FUNCTION_BLOCK p12_controlLight
VAR_INPUT
	button: BOOL;
END_VAR
VAR_OUTPUT
	light: BOOL;
END_VAR
VAR
	positiveEdgeDetection: R_TRIG;
	buttonPulse: BOOL;
	memoryCell: SR;
END_VAR

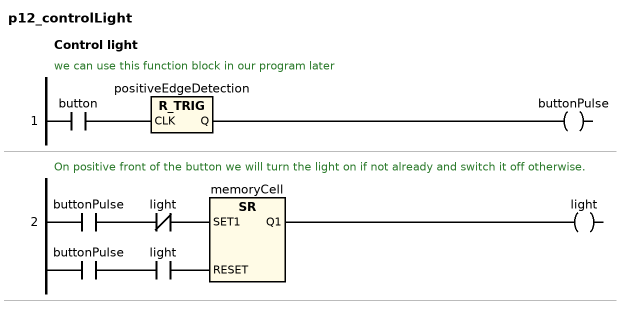
// NETWORK 1: Control light
// we can use this function block in our program later
positiveEdgeDetection(CLK := button); // R_TRIG
buttonPulse := positiveEdgeDetection.Q;

// NETWORK 2
// On positive front of the button we will turn the light on if not already and switch it off otherwise.
memoryCell(SET1 := buttonPulse AND NOT light, RESET := buttonPulse AND light); // SR
light := memoryCell.Q1;

END_FUNCTION_BLOCK

(* stored: Version 1.1.0.1, ProductVersion 3.1.4024.13
   POU p12_controlLight: Id {7a80f868-5e5a-45a7-9171-8f74fc00f7da}, SpecialFunc None *)
